FUNCTION LoadcellConvert : INT
VAR_INPUT
	LoadCellValue : INT;
END_VAR
VAR
	Voltage : REAL;
END_VAR

// Convert raw value to voltage
Voltage := INT_TO_REAL(LoadCellValue)/32767 * 10;
//convert voltage to Newtons(N) 
LoadCellConvert := REAL_TO_INT(Voltage * 980.7);

END_FUNCTION

(* stored: Version 1.1.0.1
   POU LoadcellConvert: Id {48d51865-7f04-4765-b816-c0f17f10452b}, SpecialFunc None *)
